FUNCTION_BLOCK PistonInputLogic
VAR
	timer: TOF;
	timerElapsed: BOOL;
	counter: CTU;
	id: UDINT;
	item: Item;
	location: Location;
END_VAR

timer(IN :=  NOT gvl.FotocellInput AND gvl.SwitchTablePosition, PT := T#1S, Q => timerElapsed);
counter();

IF timerElapsed AND LocalVariables.Locations[2].Item.Id = 0 THEN
	gvl.PistonInputBackwards := FALSE;
	gvl.PistonInputForward := TRUE;
	LocalVariables.Locations[2].Item.Id := LocalVariables.Locations[1].Item.Id;
	LocalVariables.Locations[2].Item.Recipe := LocalVariables.Locations[1].Item.Recipe;
	
ELSIF NOT gvl.FotocellInput THEN
	counter.CU := TRUE;
	id := counter.CV;
	LocalVariables.Locations[1].Item.Id := id;
	LocalVariables.Locations[1].Item.Recipe := LocalVariables.Recipe;

ELSE
	gvl.PistonInputBackwards := TRUE;
	gvl.PistonInputForward := FALSE;
	counter.CU := FALSE;
	LocalVariables.Locations[1].Item.Id := NULL;
END_IF

END_FUNCTION_BLOCK

(* stored: Version 1.1.0.1, ProductVersion 3.1.4024.12
   POU PistonInputLogic: Id {0374200a-6ee2-41d8-9778-4655e6023c4b}, SpecialFunc None *)
